{attribute 'qualified_only'}
VAR_GLOBAL
	Servo : AXIS_REF;
END_VAR

(* stored: Version 1.1.0.1, ProductVersion 3.1.4024.12
   GVL Motion: Id {9ee7f4e5-4f03-4067-9135-c03fe0a3f5b7} *)
